// TIA Portal project "updated for hmi 4 way" (V16)

(* hardware
DEVICE "S7-1200 station_1"  S7-1200 Station
   slot 0: "Rack_0"  S7-1200 Rack  Rack  V1.0
   slot 1: "PLC_1"  CPU 1215C DC/DC/DC  6ES7 215-1AG40-0XB0  V4.4
*)

// ===== PLC "PLC_1"  CPU 1215C DC/DC/DC =====

VAR_GLOBAL   // PLC tag table "Default tag table"
   "Input" AT %I0.1 : Bool;
   "g1" AT %Q0.2 : Bool;
   "r2" AT %Q0.3 : Bool;
   "g3" AT %Q1.0 : Bool;
   "g4" AT %Q1.3 : Bool;
   "y4" AT %Q1.2 : Bool;
   "y2" AT %Q0.4 : Bool;
   "r3" AT %Q0.6 : Bool;
   "r1" AT %Q0.0 : Bool;
   "y1" AT %Q0.1 : Bool;
   "g2" AT %Q0.5 : Bool;
   "y3" AT %Q0.7 : Bool;
   "r4" AT %Q1.1 : Bool;
   "Display" AT %M0.0 : Bool;
END_VAR

// folder: System blocks/Program resources

DATA_BLOCK "IEC_Timer_0_DB_1"   // DB2
{ S7_Optimized_Access := 'TRUE' }
AUTHOR : Simatic
FAMILY : IEC
NAME : IEC_TMR
VERSION : 1.0
// stored: InstanceOfName IEC_TIMER
"IEC_TIMER"
BEGIN
END_DATA_BLOCK

DATA_BLOCK "IEC_Timer_0_DB_2"   // DB3
{ S7_Optimized_Access := 'TRUE' }
AUTHOR : Simatic
FAMILY : IEC
NAME : IEC_TMR
VERSION : 1.0
// stored: InstanceOfName IEC_TIMER
"IEC_TIMER"
BEGIN
END_DATA_BLOCK

DATA_BLOCK "IEC_Timer_0_DB_3"   // DB4
{ S7_Optimized_Access := 'TRUE' }
AUTHOR : Simatic
FAMILY : IEC
NAME : IEC_TMR
VERSION : 1.0
// stored: InstanceOfName IEC_TIMER
"IEC_TIMER"
BEGIN
END_DATA_BLOCK

DATA_BLOCK "IEC_Timer_0_DB_4"   // DB5
{ S7_Optimized_Access := 'TRUE' }
AUTHOR : Simatic
FAMILY : IEC
NAME : IEC_TMR
VERSION : 1.0
// stored: InstanceOfName IEC_TIMER
"IEC_TIMER"
BEGIN
END_DATA_BLOCK

DATA_BLOCK "IEC_Timer_0_DB_5"   // DB6
{ S7_Optimized_Access := 'TRUE' }
AUTHOR : Simatic
FAMILY : IEC
NAME : IEC_TMR
VERSION : 1.0
// stored: InstanceOfName IEC_TIMER
"IEC_TIMER"
BEGIN
END_DATA_BLOCK

DATA_BLOCK "IEC_Timer_0_DB_6"   // DB7
{ S7_Optimized_Access := 'TRUE' }
AUTHOR : Simatic
FAMILY : IEC
NAME : IEC_TMR
VERSION : 1.0
// stored: InstanceOfName IEC_TIMER
"IEC_TIMER"
BEGIN
END_DATA_BLOCK

DATA_BLOCK "IEC_Timer_0_DB_7"   // DB8
{ S7_Optimized_Access := 'TRUE' }
AUTHOR : Simatic
FAMILY : IEC
NAME : IEC_TMR
VERSION : 1.0
// stored: InstanceOfName IEC_TIMER
"IEC_TIMER"
BEGIN
END_DATA_BLOCK

DATA_BLOCK "IEC_Timer_0_DB_8"   // DB9
{ S7_Optimized_Access := 'TRUE' }
AUTHOR : Simatic
FAMILY : IEC
NAME : IEC_TMR
VERSION : 1.0
// stored: InstanceOfName IEC_TIMER
"IEC_TIMER"
BEGIN
END_DATA_BLOCK

DATA_BLOCK "IEC_Timer_0_DB_9"   // DB10
{ S7_Optimized_Access := 'TRUE' }
AUTHOR : Simatic
FAMILY : IEC
NAME : IEC_TMR
VERSION : 1.0
// stored: InstanceOfName IEC_TIMER
"IEC_TIMER"
BEGIN
END_DATA_BLOCK

// folder: (top level)

ORGANIZATION_BLOCK "Main"   // OB1, LAD, ProgramCycle
TITLE = "Main Program Sweep (Cycle)"
{ S7_Optimized_Access := 'TRUE' }
VERSION : 0.1
BEGIN

REGION Network 1
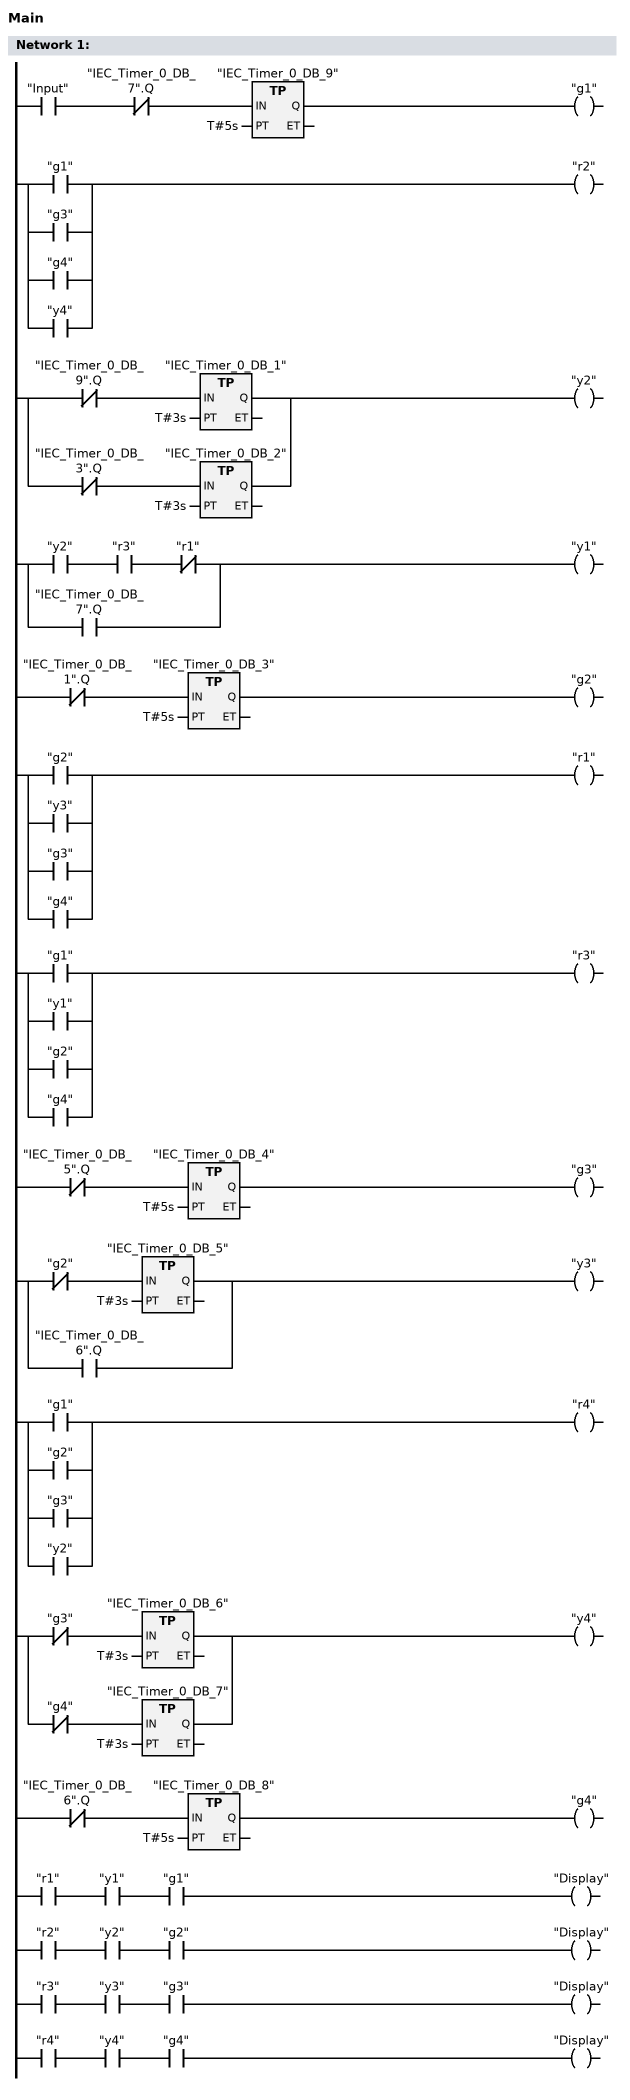
   "IEC_Timer_0_DB_9".TP(IN := "Input" AND NOT "IEC_Timer_0_DB_7".Q, PT := T#5s);
   "g1" := "IEC_Timer_0_DB_9".Q;
   "r2" := "g1" OR "g3" OR "g4" OR "y4";
   "IEC_Timer_0_DB_1".TP(IN := NOT "IEC_Timer_0_DB_9".Q, PT := T#3s);
   "IEC_Timer_0_DB_2".TP(IN := NOT "IEC_Timer_0_DB_3".Q, PT := T#3s);
   "y2" := "IEC_Timer_0_DB_1".Q OR "IEC_Timer_0_DB_2".Q;
   "y1" := ("y2" AND "r3" AND NOT "r1") OR "IEC_Timer_0_DB_7".Q;
   "IEC_Timer_0_DB_3".TP(IN := NOT "IEC_Timer_0_DB_1".Q, PT := T#5s);
   "g2" := "IEC_Timer_0_DB_3".Q;
   "r1" := "g2" OR "y3" OR "g3" OR "g4";
   "r3" := "g1" OR "y1" OR "g2" OR "g4";
   "IEC_Timer_0_DB_4".TP(IN := NOT "IEC_Timer_0_DB_5".Q, PT := T#5s);
   "g3" := "IEC_Timer_0_DB_4".Q;
   "IEC_Timer_0_DB_5".TP(IN := NOT "g2", PT := T#3s);
   "y3" := "IEC_Timer_0_DB_5".Q OR "IEC_Timer_0_DB_6".Q;
   "r4" := "g1" OR "g2" OR "g3" OR "y2";
   "IEC_Timer_0_DB_6".TP(IN := NOT "g3", PT := T#3s);
   "IEC_Timer_0_DB_7".TP(IN := NOT "g4", PT := T#3s);
   "y4" := "IEC_Timer_0_DB_6".Q OR "IEC_Timer_0_DB_7".Q;
   "IEC_Timer_0_DB_8".TP(IN := NOT "IEC_Timer_0_DB_6".Q, PT := T#5s);
   "g4" := "IEC_Timer_0_DB_8".Q;
   "Display" := "r1" AND "y1" AND "g1";
   "Display" := "r2" AND "y2" AND "g2";
   "Display" := "r3" AND "y3" AND "g3";
   "Display" := "r4" AND "y4" AND "g4";
END_REGION
END_ORGANIZATION_BLOCK